--- remSetPPS.pgx ---
program remSetPPS(string& sArgs[] (dimensions=1), string& sReturn[] (dimensions=1))
begin
  // Set the PPS status in the robot
  //
  logMsg("call remSetPPS")
  call remSetnGlobal(sArgs,nPPS,0,5000,"NOTPPS",sReturn)
end

--- remSetStagePos.pgx ---
program remSetStagePos(string& sArgs[] (dimensions=1), string& sReturn[] (dimensions=1))
begin
  // Set the PPS status in the robot
  //
  logMsg("call remSetStagePos")
  call remSetnGlobal(sArgs,nStagePos,-50000,50000,"NOTSTAGEPOS",sReturn)
end

--- remSetTCPVals.pgx ---
program remSetTCPVals(string& sArgs[] (dimensions=1), string& sReturn[] (dimensions=1))
  local bool bOk
  local num nArg
  local num nTemp
  local trsf trTCP
begin
  // Set the values of the TCP
  //
  // Arguments are "X Y Z RX RY RZ"
  //
  logMsg("call remSetTCPVals")
  nArg=0
  trTCP={0,0,0,0,0,0}
  while nArg<6
    sArgs=toNum(sArgs,nTemp,bOk)
    if bOk
      switch nArg
        case 0
          trTCP.x=nTemp
        break
        case 1
          trTCP.y=nTemp
        break
        case 2
          trTCP.z=nTemp
        break
        case 3
          trTCP.rx=nTemp
        break
        case 4
          trTCP.ry=nTemp
        break
        case 5
          trTCP.rz=nTemp
        break
      endSwitch
      nArg=nArg+1
    else
      call remErrNum("SETTCPVALS",sArgs,sReturn)
      return
    endIf
  endWhile
  tSensorTool.trsf=trTCP
  sReturn="SETTCPVALS"
end

--- remTest.pgx ---
program remTest(string& sArgs[] (dimensions=1), string& sReturn[] (dimensions=1))
  local bool bOk
  local num nAzi
  local num nEle
  local num nLoop
  local num nRX
  local num nRY
  local num nRad
  local num nVal
  local num nX
  local num nY
  local num nZ
  local string sArgsLoop
  local trsf trCalc
  local trsf trTrans
begin
  //Misc current test
  nLoop=0
  sArgsLoop=sArgs
  while nLoop<3
    sArgsLoop=toNum(sArgsLoop,nVal,bOk)
    if bOk
      switch nLoop
        case 0
          nAzi=nVal
        break
        case 1
          nEle=nVal
        break
        case 2
          nRad=nVal
        break
      endSwitch
      nLoop=nLoop+1
    else
      call remErrNum("CMDTEST",sArgs,sReturn)
      return
    endIf
  endWhile

  nZ=nRad*cos(nEle)*cos(nAzi)
  nX=nRad*cos(nEle)*sin(nAzi)
  nY=nRad*sin(nEle)
  // Decide direction det is currently facing, keep det pointed to origin
  call remCalcHereSph()
  if abs(nRXHere+nElHere)<90
    nRX=-nEle
  else
    nRX=180-nEle
  endIf
  if abs(nRYHere+nAzHere)<90
    nRY=-nAzi
  else
    nRY=180-nAzi
  endIf
  trCalc={nX,nY,nZ,nRX,nRY,nRZHere}

  trTrans={0,0,0,0,0,0}
  trTrans=trTrans*{0,0,0,0,nAzi,0}
  trTrans=trTrans*{0,0,0,-nEle,0,0}
  trTrans=trTrans*{0,0,nRad,0,0,0}
  trTrans=trTrans*{0,0,0,-180,0,0}

  putln("trCalc:  "+toString(sNumConv,trCalc.x)+" "+toString(sNumConv,trCalc.y)+" "+toString(sNumConv,trCalc.z))
  putln("         "+toString(sNumConv,trCalc.rx)+" "+toString(sNumConv,trCalc.ry)+" "+toString(sNumConv,trCalc.rz))
  putln("trTrans: "+toString(sNumConv,trTrans.x)+" "+toString(sNumConv,trTrans.y)+" "+toString(sNumConv,trTrans.z))
  putln("         "+toString(sNumConv,trTrans.rx)+" "+toString(sNumConv,trTrans.ry)+" "+toString(sNumConv,trTrans.rz))

  sReturn="No output"
end

--- remTransIP.pgx ---
program remTransIP(string& sArgs[] (dimensions=1), string& sReturn[] (dimensions=1))
  local bool bOk
  local num nLoop
  local num nVal
  local string sArgsLoop
  local trsf trUser
begin
  //Translates the current interaction point.
  //
  logMsg("call remTransIP")
  trUser={0,0,0,0,0,0}
  nLoop=0
  sArgsLoop=sArgs
  while nLoop<3
    sArgsLoop=toNum(sArgsLoop,nVal,bOk)
    if bOk
      switch nLoop
        case 0
          trUser.x=nVal
        break
        case 1
          trUser.y=nVal
        break
        case 2
          trUser.z=nVal
        break
      endSwitch
      nLoop=nLoop+1
    else
      call remErrNum("CMDTRANSIP",sArgs,sReturn)
      return
    endIf
  endWhile
  if nIPNumber==0
    fIP1.trsf=fIP1.trsf*trUser
  else
    fIP2.trsf=fIP2.trsf*trUser
  endIf
  sReturn="CMDTRANSIP"
end

--- stop.pgx ---
program stop()
begin
  //header begin
  //  PROGRAM STOP()
  //    peforms orderly shutdown functions
  //
  // initial release KN
  //header end
  //
  userPage()
  title(" SHUT DOWN ")
  cls()
  gotoxy(0,4)
  putln("WAITING:  Disabling Arm Power...")
  stopMove()
  resetMotion()
  disablePower()
  wait(isPowered()==false)
  //
  // stop tasks
  taskKill("MonitorZone")
  taskKill("RemoteControl")
  taskKill("MonitorHalt")
  taskKill("RemoteMotion")
  taskKill("iocCmdHandler")
  taskKill("RemoteMotion")
  taskKill("SimESTOP")
  //
  // tell user to press the MENU button to return to Application Menu
  cls()
  title(">>  PROGRAM STOPPED <<")
  gotoxy(0,2)
  put("Use MENU Button to return")
  gotoxy(0,3)
  put("to Main VAL3 Application Menu")
  //
  //done
end

--- tskCollision.pgx ---
program tskCollision()
  local num LnDistance
  local point LpHere
  local point LpPark
  local bool l_bPPSint
  local bool l_bStageint
  local num l_nLastChange
  local num l_nOldHeartbeat
  local num l_nTime
  local string sReturn
begin
  //header begin
  // PROGRAM tskColision()

  //header end


  do

    if dioGet(dCollisionSens)>0
      nColision=1
    else
      nColision=0
    endIf

    // logMsg(toString("",nColision))

    if dioGet(dCollisionSens)==0

      stopMove()
      resetMotion()
      disablePower()

      popUpMsg("COLLISION DETECTED!")

    endIf



  until false




end

--- tskHaltMoveMon.pgx ---
program tskHaltMoveMon()
  local bool LbZoneError
  local num LnIdx
begin
  //header begin
  // PROGRAM tskHaltMoveMon()
  //
  // This pgm is run as a separate task.
  // Will monitor if TCP Button F8 is pressed during arm motion, causes a motion stop in the initiating program.
  // Utilizes global enable bWatchForHalt==false set in pgm movTargetPoint()
  //
  //
  // incoming parms:  none
  // outgoing parms:  none
  // global parms:  bWatchForHalt => true will enable monitoring, is set in the initiating program
  //
  // called from:  pgm movTargetPoint()
  //
  //
  //  added for Release 2  KN
  //header end
  //
  // run task as infinite loop
  // initialize some bools
  bWatchForHalt=false
  do
    //
    if bWatchForHalt==true
      // while enabled, watch for F8 keypress
      // if pressed, issue bStopMotion=true
      // when bStopMotion is reset to false, then set bWatchForHalt = false and continue monitoring again
      getKey()
      while (getKey()!=278)
        delay(0)
      endWhile
      // if F8 pressed, then set the HALT MOTION global boolean
      bStopMotion=true
      wait(bWatchForHalt==false)
    endIf
    //
    delay(0)
  until (false)
end

--- tskInterlocks.pgx ---
program tskInterlocks()
  local bool l_bPPSint
  local bool l_bStageint
  local num l_nOldHeartbeat
  local num l_nLastChange
  local string sReturn
  local point LpHere
  local point LpPark
  local num LnDistance
  local num l_nTime
begin
    //header begin
  // PROGRAM tskInterlocks()
  //
  // This pgm is run as a separate task.
  // Will monitor IOC interlocks
  // Utilizes global enable bStopAllMonitor==false set in pgm mnuUtility()
  // Utilizes local enable bEnableMonitor==true set at time of motion command statement, disabled at end of motion
  //
  // Pgm will test for PPS signal while in remote mode.
  // Pgm will test for Z stage position.
  // Pgm will inform IOC of is high level mode.
  //
  // incoming parms:  none
  // outgoing parms:  none
  //
  // called from:  pgm main()
  //
  //
  //  initial release KN
  //header end
  do
    // Turn power off if door is opened and robot in remote mode
    if(nPPS <= 0 and workingMode()==4 and isPowered() )
      logMsg("Door open in remote mode. Power Disconnected")
      popUpMsg("Door open in remote mode. Power Disconnected")
      stopMove()
      resetMotion()
      disablePower()
    endIf

    // Turn off power if robot not at expected z stage position
    if(nStagePos != nStagePosOK and isPowered())
      logMsg("Robot not in correct Z stage position. Power Disconnected")
      popUpMsg("Robot not in correct Z stage position. Power Disconnected")
      stopMove()
      resetMotion()
      disablePower()
    endIf

    if(nHeartbeat !=l_nOldHeartbeat)
      l_nOldHeartbeat = nHeartbeat
      l_nLastChange = clock()
    endIf

    l_nTime = clock()-l_nLastChange

    // Turn off power if robot looses connection to IOC in remote mode
    if(workingMode()==4 and isPowered())
      if(l_nTime>2)
        stopMove()
        resetMotion()
        disablePower()

        logMsg("Lost IOC hearbeat! Power Disconnected")
        sReturn="ERROR 902"
        sReturn=sReturn+": Lost IOC hearbeat! Power Disconnected. "+(toString(".4",l_nTime))
        putln(sReturn)
        logMsg(sReturn)

      endIf
      endIf

    // Report the high level robot mode
    // 0 - Not Parker
    // 1 - Parked
    // 2 - Parked Top

    nRobotMode = 0

    LpHere=here(tSensorTool,world)
    LpPark=jointToPoint(tSensorTool,world,jPark)
    LnDistance=abs(distance(LpHere,LpPark))
    if LnDistance<=nParkTolerance
      nRobotMode = 1
    endIf

    LpHere=here(tSensorTool,world)
    LpPark=jointToPoint(tSensorTool,world,jParkTop)
    LnDistance=abs(distance(LpHere,LpPark))
    if LnDistance<=nParkTolerance
      nRobotMode = 2
    endIf


    delay(0.1)



  until false




end

--- tskMonitorZone.pgx ---
program tskMonitorZone()
  local bool LbZoneError
  local num LnIdx
begin
  //header begin
  // PROGRAM tskMonitorZone()
  //
  // This pgm is run as a separate task.
  // Will monitor if TCP is in a Stay Clear Zone during arm motion.
  // Utilizes global enable bStopAllMonitor==false set in pgm mnuUtility()
  // Utilizes local enable bEnableMonitor==true set at time of motion command statement, disabled at end of motion
  //
  // Pgm will test for TCP inside a defined "Stay Clear Zone" during moves.
  //
  // Zones are defined if MON:bCreateCube[nIndex], MON:bCreateCylinder[nIndex], MON:bCreateSphere[nIndex] are true, ...
  // these bools are set at time of teaching or set explicitly
  // If TCP enters a defined zone, then a boolean is set and motion is stopped immediately at the motion program.
  //
  // incoming parms:  none
  // outgoing parms:  none
  // global parms:  bEnableMonitor => true will enable monitoring, is set before each required...
  //                                  move statement
  //                bStopAllMonitor => false will allow monitor, is a MASTER level...
  //                                   boolean set in pgm mnuUtility()
  //
  // called from:  pgm main()
  //
  // argument descriptions for zone check calls are found in library "monitorAreaEn"
  //
  //  initial release KN
  //header end
  //
  // run task as infinite loop
  // initialize some bools, these are reset in pgm movTargetPoint() or when bStopAllMonitor=true (set in pgm mnuUtility() )
  bInsideCube=false
  bInsideCylinder=false
  bInsideSphere=false
  LbZoneError=false
  do
    //
    // CONDITION 1of2:  Master Zone Monitor Enable/Disable
    if (bStopAllMonitor==false)
      // CONDITION 2of2:  run the zone checks if the "while in motion" boolean bEnableMonitor is enabled
      if (bEnableMonitor==true)
        // put "Zone Monitoring enabled" indicator at a discreet location on MPC screen
        gotoxy(39,13)
        put("M")
        //
        for LnIdx=0 to 9
          // verify if cube zone defined, test tSensorTool location
          if MON:bCreateCube[LnIdx]==true
            call MON:checkCube(tSensorTool,LnIdx,bInsideCube,LbZoneError)
          endIf
          // verify cylinder zone defined, test tSensorTool location
          if MON:bCreateCylinder[LnIdx]==true
            call MON:checkCylinder(tSensorTool,LnIdx,bInsideCylinder,LbZoneError)
          endIf
          // verify sphere zone defined, test tSensorTool location
          if MON:bCreateSphere[LnIdx]==true
            call MON:checkSphere(tSensorTool,LnIdx,bInsideSphere,LbZoneError)
          endIf
          delay(0)
        endFor
        //
      endIf
    else
      bInsideCube=false
      bInsideCylinder=false
      bInsideSphere=false
    endIf
    //
    delay(0)
  until (false)
end

--- tskRemControl1.pgx ---
program tskRemControl1()
  local bool LbError
  local bool LbRemControlEnd
  local bool LbRemoteDone
  local num LnIdx
  local num LnLoginCounter
  local num LnTimerStart
  local num LnTimerValue
  local string LsCommandString
  local string LsCubeValsIOC
  local string LsCylValsIOC
  local string LsESTOPIOC
  local string LsError
  local string LsJointValsIOC
  local string LsLength
  local string LsResponse
  local string LsSphValsIOC
  local string LsTCPValsIOC
begin
  // PROGRAM tskRemControl1()
  //
  // Accepts commands sent from IOC and responds accordingly.
  // This program will always be running in a "read-only" mode, where we
  // allow only commands that begin with "GET" as well as "ENABLEREMOTE"
  //
  // We can switch to the "write-enabled" mode from the MCP or by sending
  // "ENABLEREMOTE". We can switch back to the "read-only" mode (MANUAL)
  // by sending "HALTREMOTE" or by pressing 1 on the MCP.
  //
  // Commands are of the form "CMD ARG1 ARG2 ARG3..." and respond with
  // "CMD VAL1 VAL2 VAL3...", or instead with "ERROR ###: Text" if something
  // goes wrong.
  //
  // start infinite loop
  do
    // start remCmdHandler with bRemControlON=false for limit to get commands and no putln
    if taskStatus("iocCmdHandler")!=1
      if (taskStatus("iocCmdHandler")==125)
        logMsg("read-only iocCmdHandler dead, restarting...")
        taskKill("iocCmdHandler")
        wait(taskStatus("iocCmdHandler")==-1)
        clearBuffer(sioIOCclient)
      endIf
      logMsg("start remCmdHandler for passive commands...")
      taskCreate "iocCmdHandler",30,remCmdHandler()
      wait(taskStatus("iocCmdHandler")==1)
    endIf
    //
    // bRemControlON set in pgm mnuUtility()
    if bRemControlON==true
      userPage()
      cls()
      title(" REMOTE CONTROL REQUESTED ")
      // test for ESTOP, request action if active
      if esStatus()!=0
        gotoxy(0,4)
        putln("WAITING:  Reset ESTOP")
        wait(esStatus()==0)
      endIf
      //
      // setup user page & open IOC via ethernet socket as CS8 Server socket connection
      userPage()
      cls()
      title(" REMOTE CONTROL ACTIVE ")
      cls()
      putln("Start Remote Control, arm power OFF")
      logMsg("Start Remote Control, arm power OFF")
      bKillRemControl=false
      // bKillRemControl is set in tskCmdHandler() and reacted to in following do-until loop
      if taskStatus("iocCmdHandler")!=1
        logMsg("iocCmdHandler task OFF, starting...")
        putln("IOC Cmd Handler task OFF, starting...")
        taskCreate "iocCmdHandler",30,remCmdHandler()
        wait(taskStatus("iocCmdHandler")==1)
      endIf
      logMsg("iocCmdHandler active now")
      putln("IOC Command Handler task ON")

      // Test for simulated ESTOP
      if bSimulateESTOP==true
        if taskStatus("SimESTOP")==-1
          taskCreate "SimESTOP",35,tskSimESTOP()
          wait(taskStatus("SimESTOP")==1)
        endIf
      endIf
      bSimESTOPOn=false

      wait(taskStatus("RemoteMotion")==1)
      putln(" ")
      putln("LISTENING for IOC Client now...")
      logMsg("listening IOC now")
      LbRemControlEnd=false
      do
        // monitor ESTOP status during remote control, manage restart if needed
        if esStatus()!=0 or bSimESTOPOn==true
          cls()
          putln("ESTOP ESTOP ESTOP ESTOP")
          logMsg("FAULT:  ESTOP!")
          call iocWriteBack("ESTOPSTATX"+" "+toString(".0",esStatus()))
          logMsg("kill tskRemMotion on ESTOP")
          putln("kill Remote Motion task on ESTOP")
          sIOCCommand=""
          sRemMotionCmd=""
          taskKill("RemoteMotion")
          wait(taskStatus("RemoteMotion")!=1)
          logMsg("tskRemMotion killed on ESTOP")
          putln("Remote Motion task killed on ESTOP")
          stopMove()
          resetMotion()
          disablePower()
          wait(isPowered()==false)
          bRemMotionBusy=false
          //
          putln("")
          if bSimulateESTOP==true
            putln("delay 5 sec for ESTOP RESET")
            delay(5)
            putln("sim ESTOP RESET done, CONTINUE")
            bSimESTOPOn=false
          else
            putln("WAITING:  reset ESTOP")
            logMsg("WAITING:  reset ESTOP")
            wait(esStatus()==0)
            putln("ESTOP has been RESET!")
            logMsg("ESTOP has been RESET!")
          endIf
          putln("")
        endIf
        //
        // monitor bKillRemControl set in tskCmdHandler, stop tskCmdHandler if needed
        if bKillRemControl==true
          //call iocWriteBack("REMOTEHALT")
          putln("IOC requested HALT REMOTE CONTROL")
          logMsg("IOC requested HALT REMOTE CONTROL")
          stopMove()
          resetMotion()
          bRemMotionBusy=false
          //
          // kill Remote Motion task
          bRemControlON=false
          putln("STOPPING RemoteMotion task...")
          logMsg("STOPPING RemoteMotion task...")
          taskKill("RemoteMotion")
          wait(taskStatus("RemoteMotion")!=1)
          putln("RemoteMotion task STOPPED!")
          logMsg("RemoteMotion task STOPPED!")
          LbRemControlEnd=true
          //
          if bSimulateESTOP==true
            // kill ESTOP Simulation task
            putln("STOPPING ESTOP Simulator task...")
            logMsg("STOPPING ESTOP Simulator task...")
            taskKill("SimESTOP")
            wait(taskStatus("SimESTOP")!=1)
            putln("ESTOP Simulator task STOPPED!")
            logMsg("ESTOP Similator task STOPPED!")
          endIf
        endIf

        // Code adapted from Jan Meyer to reopen socket in the event that iocCmdHandler hangs
        // works by checking if taskStatus("iocCmdHandler")==125 (Read or write error on a dio, aio, sio)
        if (taskStatus("iocCmdHandler")!=1 and taskStatus("iocCmdHandler")!=-1)
          // reopen socket on error
          if (taskStatus("iocCmdHandler")==125)
            putln("R/W error on sioIOCclient")
            putln("Killing iocCmdHandler")
            taskKill("iocCmdHandler")
            wait(taskStatus("iocCmdHandler")==-1)
            putln("iocCmdHandler dead. Restarting...")
            clearBuffer(sioIOCclient)
            logMsg("iocCmdHandler task OFF, starting...")
            taskCreate "iocCmdHandler",30,remCmdHandler()
            wait(taskStatus("iocCmdHandler")==1)
            logMsg("iocCmdHandler active now")
            putln("IOC Command Handler task ON")
          endIf
        endIf

        delay(0)
      until LbRemControlEnd==true
      putln("")
      //
      cls()
      title(" MANUAL CONTROL REQUESTED ")
      gotoxy(0,4)
      putln("WAITING:  Arm Power Disable")
      disablePower()
      wait(isPowered()==false)
      cls()
      gotoxy(0,4)
      putln("WAITING:  Change to MANUAL MODE")
      wait(workingMode()==1)
      cls()
      gotoxy(0,4)
      putln("  Press ESC to return to manual menu.")
    endIf
    //
    delay(0)
  until false
  //
  //done
end

--- tskSimESTOP.pgx ---
program tskSimESTOP()
  local num LnKey
begin
  bSimESTOPOn=false
  LnKey=1111
  do
    LnKey=getKey()
    // test if Function button F1->F8 is pressed on Emulator
    if bSimESTOPOn==false and (LnKey==271 or LnKey==272 or LnKey==273 or LnKey==274 or LnKey==275 or LnKey==276 or LnKey==277 or LnKey==278)
      bSimESTOPOn=true
      putln("Simulated ESTOP")
      delay(1)
      LnKey=1111
    endIf
    delay(0)
  until false
end

--- xppWriteBack.pgx ---
program xppWriteBack(string XsResponse (dimensions=1))
begin
  //
  //header begin
  // PROGRAM xppWriteBack()
  //
  // pgm writes text via TCP/IP to XPP client socket on CS8
  //
  // input parms:
  //    XsResponse = string passed from calling program
  //
  // output parms:
  //    none
  //
  // called from:  xppCmdHandler()
  //
  // initial release:  KN
  // Release 2:  KN
  //  changed functionality from CS8 host to CS8 client
  //  updated documentation
  //header end
  //
  sioXPPclient=XsResponse
end
